// TIA Portal V17 export
// export: Created 2023-12-22T15:28:34.8526887Z, ExportSetting WithDefaults, DisplayName Totally Integrated Automation Portal, DisplayVersion V17, DisplayName TIA Portal Openness, DisplayVersion V17, DisplayName TIA Portal Version Control Interface, DisplayVersion V17, DisplayName STEP 7 Professional, DisplayVersion V17, DisplayName STEP 7 Safety, DisplayVersion V17, DisplayName WinCC Advanced, DisplayVersion V17
FUNCTION_BLOCK "DRV_V_D2A"   // FB121, LAD
TITLE = Управление клапаном с двумя дискретными положениями
{ S7_Optimized_Access := 'FALSE' }
VERSION : 0.1
// stored: AutoNumber false, IsIECCheckEnabled false, SetENOAutomatically false, UDAEnableTagReadback false
   VAR_INPUT
      All_Block : Bool;   // Аварийный останов
   END_VAR
   VAR_IN_OUT
      FB_QF : Bool;   // Защитный автомат
      FB_KM_Open : Bool;   // Пускатель - открыть
      FB_KM_Close : Bool;   // Пускатель - закрыть
      FB_Open : Bool;   // ОС - открыто
      FB_Close : Bool;   // ОС - закрыто
      S_Alarm : Bool;   // Наличие аварии
      CMD_Open : Bool;   // Команда - открыть
      CMD_Close : Bool;   // Команда - закрыть
   END_VAR
   VAR DB_SPECIFIC
      CMD : "CMD";   // Блок команд
      Mode : Int;   // Режим работы
      Status : Int;   // Статус устройства
      Use : Struct   // Функционал
         QF { S7_SetPoint := 'True'} : Bool;   // Защитный автомат
         KM_Open { S7_SetPoint := 'True'} : Bool;   // Пускатель - открыть
         KM_Close { S7_SetPoint := 'True'} : Bool;   // Пускатель - закрыть
         Open { S7_SetPoint := 'True'} : Bool := true;   // ОС - открыто
         Close { S7_SetPoint := 'True'} : Bool := true;   // ОС - закрыто
         One_KM { S7_SetPoint := 'True'} : Bool;   // Общий пускатель
         Electro { S7_SetPoint := 'True'} : Bool;   // Электропривод (остановка при срабатывании концевика)
         Cross { S7_SetPoint := 'True'} : Bool;   // Кросс-замена датчиков
         CMD_Open { S7_SetPoint := 'True'} : Bool := true;
         CMD_Close { S7_SetPoint := 'True'} : Bool;
         CMD_Reset { S7_SetPoint := 'True'} : Bool;
         calibration : Bool;
      END_STRUCT;
      FB : Struct   // Функционал
         Ready : Bool;   // Готовность к запуску
         QF : Bool;   // Защитный автомат
         KM_Open : Bool;   // Пускатель - открыть
         KM_Close : Bool;   // Пускатель - закрыть
         Open : Bool;   // ОС - открыто
         Close : Bool;   // ОС - закрыто
         Reserv : Bool;
         Local_Open : Bool;   // Локальное открытие
         Local_Close : Bool;   // Локальное закрытие
         pos_ok : Bool;   // положение достигнуто
         pos_open : Bool;   // клапан открывается
         pos_close : Bool;   // клапан закрывается
      END_STRUCT;
      ON : Bool;   // Успешно запущено
      OFF : Bool;   // Успешно остановлено
      REQ_Open : Bool;   // Запрос на открытие
      REQ_Close : Bool;   // Запрос на закрытие
   END_VAR
   VAR
      Tx { S7_SetPoint := 'True'} : Array[0..4] of "Time_S";   // Блок таймеров
   END_VAR
   VAR DB_SPECIFIC
      Inv : Struct   // Инверсия сигналов
         CMD { S7_SetPoint := 'True'} : Bool;   // Команда запуска
         QF { S7_SetPoint := 'True'} : Bool;   // Защитный автомат
         KM_Open { S7_SetPoint := 'True'} : Bool;   // Пускатель - открыть
         KM_Close { S7_SetPoint := 'True'} : Bool;   // Пускатель - закрыть
         Serivce { S7_SetPoint := 'True'} : Bool;   // Сервисный выключатель
         Open { S7_SetPoint := 'True'} : Bool;   // ОС - открыто
         Close { S7_SetPoint := 'True'} : Bool;   // ОС - закрыто
         Local_Open { S7_SetPoint := 'True'} : Bool;   // Локальное открытие
         Local_Close { S7_SetPoint := 'True'} : Bool;   // Локальное закрытие
      END_STRUCT;
      Alarm : Struct   // Список аварий
         Block : Bool;   // Аварийная остановка
         QF : Bool;   // Выбило защитный автомат
         KM_Open : Bool;   // Не сработал пускатель - открыть
         KM_Close : Bool;   // Не сработал пускатель - закрыть
         Two_S : Bool;   // Две ОС
         Open : Bool;   // Не сработал концевик - открыто
         Close : Bool;   // Не сработал концевик - закрыто
         OpTime : Bool;
      END_STRUCT;
      Alarms : Word;   // Слово аварий
      OpTime_h : DInt;   // наработка (ч)
      OpTime_s { S7_SetPoint := 'True'} : DInt;   // наработка (с)
      CodeID { S7_SetPoint := 'True'} : Int;   // Код датчика для привязки в скаде
      Indirect : Struct
         FB_QF { S7_SetPoint := 'True'} : Bool := true;   // Защитный автомат
         FB_KM_Open { S7_SetPoint := 'True'} : Bool := true;   // Пускатель - открыть
         FB_KM_Close { S7_SetPoint := 'True'} : Bool := true;   // Пускатель - закрыть
         FB_Open { S7_SetPoint := 'True'} : Bool := true;   // ОС - открыто
         FB_Close { S7_SetPoint := 'True'} : Bool := true;   // ОС - закрыто
         CMD_Open { S7_SetPoint := 'True'} : Bool := true;   // Команда на открытие
         CMD_Close { S7_SetPoint := 'True'} : Bool := true;   // Команда на закрытие
      END_STRUCT;
      Indirect_BYTE : Struct
         FB_QF { S7_SetPoint := 'True'} : Int;   // Защитный автомат
         FB_KM_Open { S7_SetPoint := 'True'} : Int;   // Пускатель - открыть
         FB_KM_Close { S7_SetPoint := 'True'} : Int;   // Пускатель - закрыть
         FB_Open { S7_SetPoint := 'True'} : Int;   // ОС - открыто
         FB_Close { S7_SetPoint := 'True'} : Int;   // ОС - закрыто
         CMD_Open { S7_SetPoint := 'True'} : Int;   // Команда на открытие
         CMD_Close { S7_SetPoint := 'True'} : Int;   // Команда на закрытие
         CMD_Reset : Int;
      END_STRUCT;
      Indirect_BIT : Struct
         FB_QF { S7_SetPoint := 'True'} : Int;   // Защитный автомат
         FB_KM_Open { S7_SetPoint := 'True'} : Int;   // Пускатель - открыть
         FB_KM_Close { S7_SetPoint := 'True'} : Int;   // Пускатель - закрыть
         FB_Open { S7_SetPoint := 'True'} : Int;   // ОС - открыто
         FB_Close { S7_SetPoint := 'True'} : Int;   // ОС - закрыто
         CMD_Open { S7_SetPoint := 'True'} : Int;   // Команда на открытие
         CMD_Close { S7_SetPoint := 'True'} : Int;   // Команда на закрытие
         CMD_Reset : Int;
      END_STRUCT;
   END_VAR
   VAR
      Tx_Sm { S7_SetPoint := 'True'} : Array[0..2] of "Time_S_b";   // Блок таймеров
      Tx_R { S7_SetPoint := 'True'} : Array[0..1] of "Time_R";   // Блок таймеров
   END_VAR
   VAR DB_SPECIFIC
      SP_A : Real;
      SP_M : Real;
      SP : Real;
      POSITION : Real;
      "step" : Int;
      DB { S7_SetPoint := 'True'} : Real := 1.0;
      pos : Array[0..15] of Bool;
   END_VAR
   VAR_TEMP
      xQF : Bool;
      xKM_Open : Bool;
      xKM_Close : Bool;
      xOpen : Bool;
      xClose : Bool;
      min : Real;
      max : Real;
   END_VAR
   VAR CONSTANT
      Pos_MIN : Real := 0.0;
      Pos_MAX : Real := 100.0;
   END_VAR
   VAR_TEMP   // added for the SCL form of the ladder/FBD networks
      _w1 : Bool;
      _w2 : Bool;
      _w3 : Bool;
      _w4 : Bool;
      _w5 : Bool;
      _w6 : Bool;
      _w7 : Bool;
   END_VAR
BEGIN

REGION Network 1: Режим глобальной симуляции
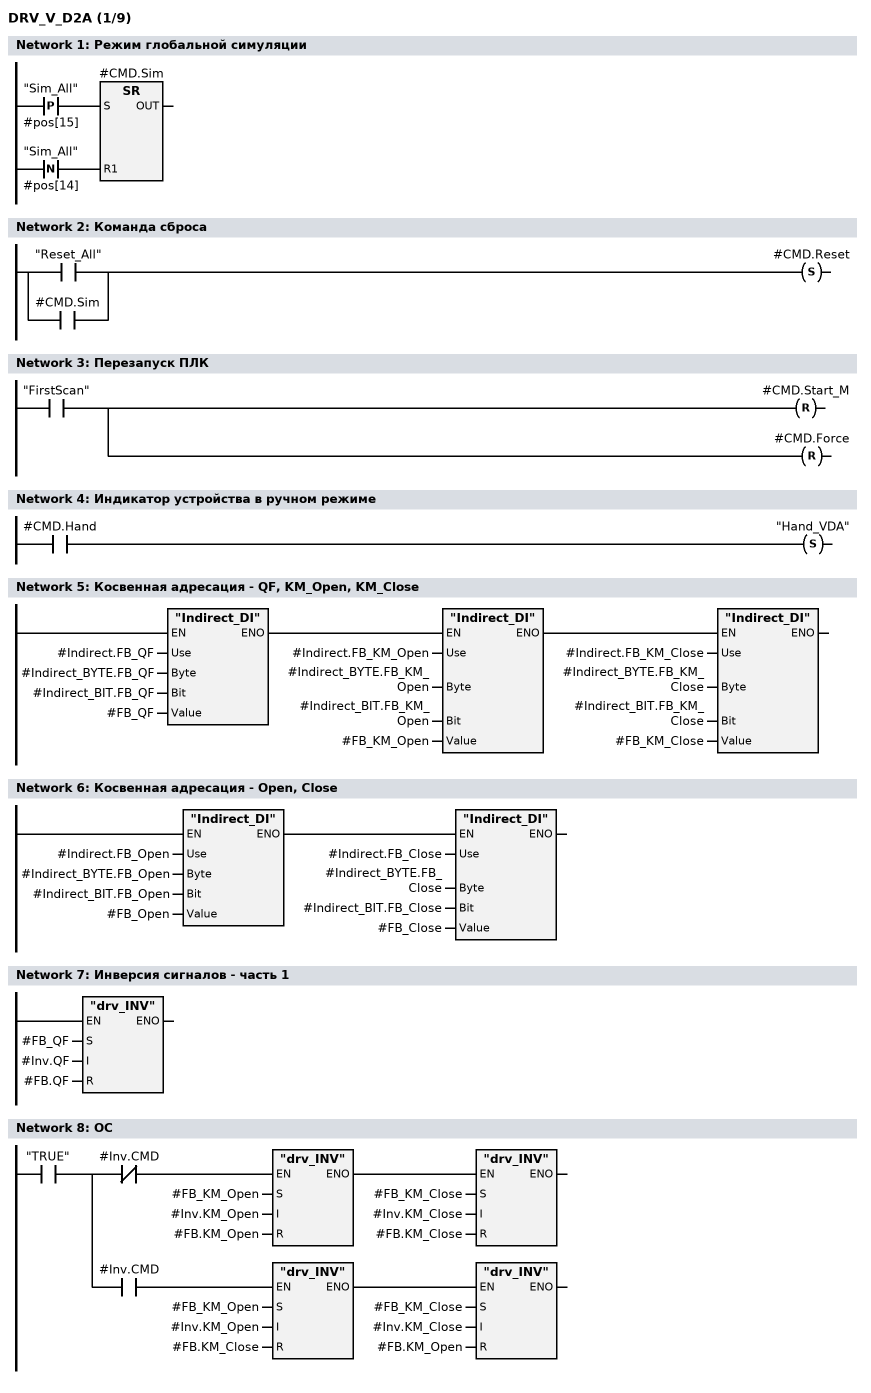
   RUNG wire#powerrail
      P_Contact(operand := "Sim_All", bit := #pos[15])
      S_SR(operand := #CMD.Sim, r1 := wire#w1)
   END_RUNG
   RUNG wire#powerrail
      N_Contact(operand := "Sim_All", bit := #pos[14])
   END_RUNG wire#w1
   // the same network as SCL:
   #_w1 := "Sim_All" AND NOT #pos[15];   // rising edge of "Sim_All"
   #pos[15] := "Sim_All";
   #_w2 := NOT "Sim_All" AND #pos[14];   // falling edge of "Sim_All"
   #pos[14] := "Sim_All";
   IF #_w1 THEN
       #CMD.Sim := TRUE;   // SR flip-flop
   END_IF;
   IF #_w2 THEN #CMD.Sim := FALSE; END_IF;
END_REGION

REGION Network 2: Команда сброса
   RUNG wire#powerrail
      Contact( "Reset_All" )
      wire#w1
      S_Coil( #CMD.Reset )
   END_RUNG
   RUNG wire#powerrail
      Contact( #CMD.Sim )
   END_RUNG wire#w1
   // the same network as SCL:
   IF "Reset_All" OR #CMD.Sim THEN #CMD.Reset := TRUE; END_IF;
END_REGION

REGION Network 3: Перезапуск ПЛК
   RUNG wire#powerrail
      Contact( "FirstScan" )
      wire#w1
      R_Coil( #CMD.Start_M )
   END_RUNG
   RUNG wire#w1
      R_Coil( #CMD.Force )
   END_RUNG
   // the same network as SCL:
   IF "FirstScan" THEN
       #CMD.Start_M := FALSE;
       #CMD.Force := FALSE;
   END_IF;
END_REGION

REGION Network 4: Индикатор устройства в ручном режиме
   RUNG wire#powerrail
      Contact( #CMD.Hand )
      S_Coil( "Hand_VDA" )
   END_RUNG
   // the same network as SCL:
   IF #CMD.Hand THEN "Hand_VDA" := TRUE; END_IF;
END_REGION

REGION Network 5: Косвенная адресация - QF, KM_Open, KM_Close
   RUNG wire#powerrail
      "Indirect_DI"(Use := #Indirect.FB_QF, "Byte" := #Indirect_BYTE.FB_QF, Bit := #Indirect_BIT.FB_QF, Value := #FB_QF)
      "Indirect_DI"(Use := #Indirect.FB_KM_Open, "Byte" := #Indirect_BYTE.FB_KM_Open, Bit := #Indirect_BIT.FB_KM_Open, Value := #FB_KM_Open)
      "Indirect_DI"(Use := #Indirect.FB_KM_Close, "Byte" := #Indirect_BYTE.FB_KM_Close, Bit := #Indirect_BIT.FB_KM_Close, Value := #FB_KM_Close)
   END_RUNG
   // the same network as SCL:
   "Indirect_DI"(Use := #Indirect.FB_QF,
                 "Byte" := #Indirect_BYTE.FB_QF,
                 Bit := #Indirect_BIT.FB_QF,
                 Value := #FB_QF,
                 ENO => #_w1);
   "Indirect_DI"(EN := #_w1,
                 Use := #Indirect.FB_KM_Open,
                 "Byte" := #Indirect_BYTE.FB_KM_Open,
                 Bit := #Indirect_BIT.FB_KM_Open,
                 Value := #FB_KM_Open,
                 ENO => #_w2);
   IF #_w2 THEN
       "Indirect_DI"(Use := #Indirect.FB_KM_Close,
                     "Byte" := #Indirect_BYTE.FB_KM_Close,
                     Bit := #Indirect_BIT.FB_KM_Close,
                     Value := #FB_KM_Close);
   END_IF;
END_REGION

REGION Network 6: Косвенная адресация - Open, Close
   RUNG wire#powerrail
      "Indirect_DI"(Use := #Indirect.FB_Open, "Byte" := #Indirect_BYTE.FB_Open, Bit := #Indirect_BIT.FB_Open, Value := #FB_Open)
      "Indirect_DI"(Use := #Indirect.FB_Close, "Byte" := #Indirect_BYTE.FB_Close, Bit := #Indirect_BIT.FB_Close, Value := #FB_Close)
   END_RUNG
   // the same network as SCL:
   "Indirect_DI"(Use := #Indirect.FB_Open,
                 "Byte" := #Indirect_BYTE.FB_Open,
                 Bit := #Indirect_BIT.FB_Open,
                 Value := #FB_Open,
                 ENO => #_w1);
   IF #_w1 THEN
       "Indirect_DI"(Use := #Indirect.FB_Close,
                     "Byte" := #Indirect_BYTE.FB_Close,
                     Bit := #Indirect_BIT.FB_Close,
                     Value := #FB_Close);
   END_IF;
END_REGION

REGION Network 7: Инверсия сигналов - часть 1
   RUNG wire#powerrail
      "drv_INV"(S := #FB_QF, I := #Inv.QF, R := #FB.QF)
   END_RUNG
   // the same network as SCL:
   "drv_INV"(S := #FB_QF, I := #Inv.QF, R := #FB.QF);
END_REGION

REGION Network 8: ОС
   RUNG wire#powerrail
      Contact( "TRUE" )
      wire#w1
      I_Contact( #Inv.CMD )
      "drv_INV"(S := #FB_KM_Open, I := #Inv.KM_Open, R := #FB.KM_Open)
      "drv_INV"(S := #FB_KM_Close, I := #Inv.KM_Close, R := #FB.KM_Close)
   END_RUNG
   RUNG wire#w1
      Contact( #Inv.CMD )
      "drv_INV"(S := #FB_KM_Open, I := #Inv.KM_Open, R := #FB.KM_Close)
      "drv_INV"(S := #FB_KM_Close, I := #Inv.KM_Close, R := #FB.KM_Open)
   END_RUNG
   // the same network as SCL:
   #_w2 := "TRUE";
   "drv_INV"(EN := "TRUE" AND NOT #Inv.CMD, S := #FB_KM_Open, I := #Inv.KM_Open, R := #FB.KM_Open, ENO => #_w1);
   IF #_w1 THEN "drv_INV"(S := #FB_KM_Close, I := #Inv.KM_Close, R := #FB.KM_Close); END_IF;
   "drv_INV"(EN := #_w2 AND #Inv.CMD, S := #FB_KM_Open, I := #Inv.KM_Open, R := #FB.KM_Close, ENO => #_w3);
   IF #_w3 THEN "drv_INV"(S := #FB_KM_Close, I := #Inv.KM_Close, R := #FB.KM_Open); END_IF;
END_REGION

REGION Network 9: Инверсия сигналов - часть 2
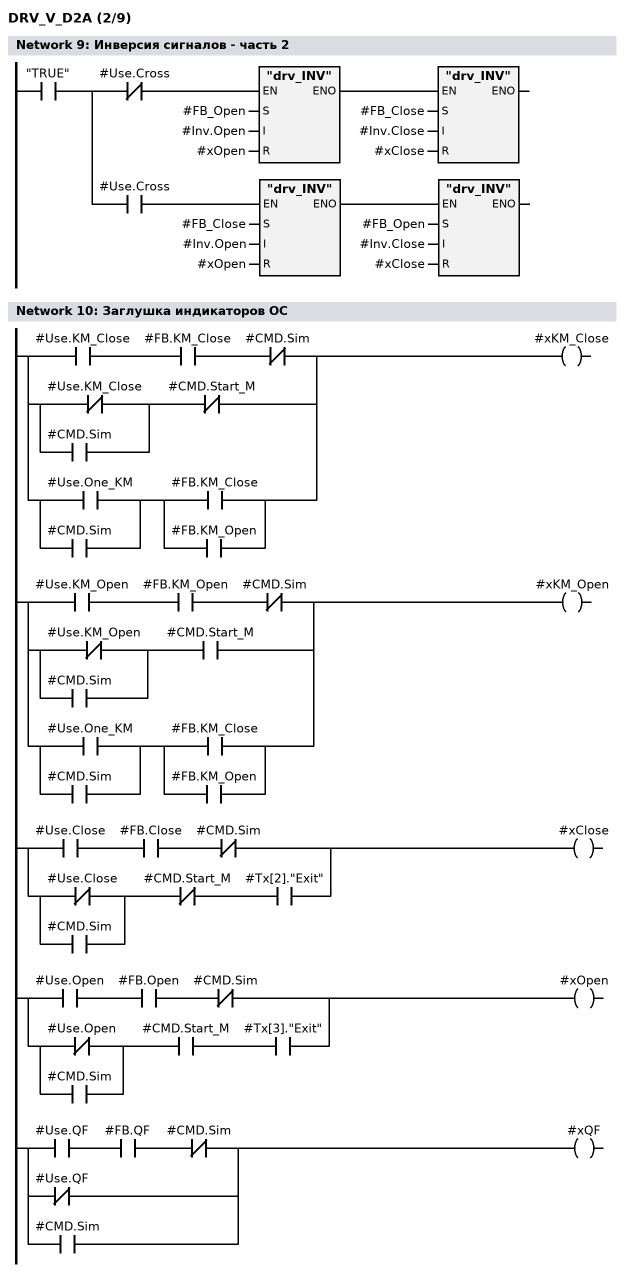
   RUNG wire#powerrail
      Contact( "TRUE" )
      wire#w1
      I_Contact( #Use.Cross )
      "drv_INV"(S := #FB_Open, I := #Inv.Open, R := #xOpen)
      "drv_INV"(S := #FB_Close, I := #Inv.Close, R := #xClose)
   END_RUNG
   RUNG wire#w1
      Contact( #Use.Cross )
      "drv_INV"(S := #FB_Close, I := #Inv.Open, R := #xOpen)
      "drv_INV"(S := #FB_Open, I := #Inv.Close, R := #xClose)
   END_RUNG
   // the same network as SCL:
   #_w2 := "TRUE";
   "drv_INV"(EN := "TRUE" AND NOT #Use.Cross, S := #FB_Open, I := #Inv.Open, R := #xOpen, ENO => #_w1);
   IF #_w1 THEN "drv_INV"(S := #FB_Close, I := #Inv.Close, R := #xClose); END_IF;
   "drv_INV"(EN := #_w2 AND #Use.Cross, S := #FB_Close, I := #Inv.Open, R := #xOpen, ENO => #_w3);
   IF #_w3 THEN "drv_INV"(S := #FB_Open, I := #Inv.Close, R := #xClose); END_IF;
END_REGION

REGION Network 10: Заглушка индикаторов ОС
   RUNG wire#powerrail
      Contact( #Use.KM_Close )
      Contact( #FB.KM_Close )
      I_Contact( #CMD.Sim )
      wire#w1
      Coil( #xKM_Close )
   END_RUNG
   RUNG wire#powerrail
      I_Contact( #Use.KM_Close )
      wire#w2
      I_Contact( #CMD.Start_M )
   END_RUNG wire#w1
   RUNG wire#powerrail
      Contact( #CMD.Sim )
   END_RUNG wire#w2
   RUNG wire#powerrail
      Contact( #Use.One_KM )
      wire#w3
      Contact( #FB.KM_Close )
   END_RUNG wire#w1
   RUNG wire#powerrail
      Contact( #CMD.Sim )
   END_RUNG wire#w3
   RUNG wire#w3
      Contact( #FB.KM_Open )
   END_RUNG wire#w1
   RUNG wire#powerrail
      Contact( #Use.KM_Open )
      Contact( #FB.KM_Open )
      I_Contact( #CMD.Sim )
      wire#w4
      Coil( #xKM_Open )
   END_RUNG
   RUNG wire#powerrail
      I_Contact( #Use.KM_Open )
      wire#w5
      Contact( #CMD.Start_M )
   END_RUNG wire#w4
   RUNG wire#powerrail
      Contact( #CMD.Sim )
   END_RUNG wire#w5
   RUNG wire#powerrail
      Contact( #Use.One_KM )
      wire#w6
      Contact( #FB.KM_Close )
   END_RUNG wire#w4
   RUNG wire#powerrail
      Contact( #CMD.Sim )
   END_RUNG wire#w6
   RUNG wire#w6
      Contact( #FB.KM_Open )
   END_RUNG wire#w4
   RUNG wire#powerrail
      Contact( #Use.Close )
      Contact( #FB.Close )
      I_Contact( #CMD.Sim )
      wire#w7
      Coil( #xClose )
   END_RUNG
   RUNG wire#powerrail
      I_Contact( #Use.Close )
      wire#w8
      I_Contact( #CMD.Start_M )
      Contact( #Tx[2]."Exit" )
   END_RUNG wire#w7
   RUNG wire#powerrail
      Contact( #CMD.Sim )
   END_RUNG wire#w8
   RUNG wire#powerrail
      Contact( #Use.Open )
      Contact( #FB.Open )
      I_Contact( #CMD.Sim )
      wire#w9
      Coil( #xOpen )
   END_RUNG
   RUNG wire#powerrail
      I_Contact( #Use.Open )
      wire#w10
      Contact( #CMD.Start_M )
      Contact( #Tx[3]."Exit" )
   END_RUNG wire#w9
   RUNG wire#powerrail
      Contact( #CMD.Sim )
   END_RUNG wire#w10
   RUNG wire#powerrail
      Contact( #Use.QF )
      Contact( #FB.QF )
      I_Contact( #CMD.Sim )
      wire#w11
      Coil( #xQF )
   END_RUNG
   RUNG wire#powerrail
      I_Contact( #Use.QF )
   END_RUNG wire#w11
   RUNG wire#powerrail
      Contact( #CMD.Sim )
   END_RUNG wire#w11
   // the same network as SCL:
   #xKM_Close := (#Use.KM_Close AND #FB.KM_Close AND NOT #CMD.Sim) OR ((NOT #Use.KM_Close OR #CMD.Sim) AND NOT #CMD.Start_M) OR ((#Use.One_KM OR #CMD.Sim) AND (#FB.KM_Close OR #FB.KM_Open));
   #xKM_Open := (#Use.KM_Open AND #FB.KM_Open AND NOT #CMD.Sim) OR ((NOT #Use.KM_Open OR #CMD.Sim) AND #CMD.Start_M) OR ((#Use.One_KM OR #CMD.Sim) AND (#FB.KM_Close OR #FB.KM_Open));
   #xClose := (#Use.Close AND #FB.Close AND NOT #CMD.Sim) OR ((NOT #Use.Close OR #CMD.Sim) AND NOT #CMD.Start_M AND #Tx[2]."Exit");
   #xOpen := (#Use.Open AND #FB.Open AND NOT #CMD.Sim) OR ((NOT #Use.Open OR #CMD.Sim) AND #CMD.Start_M AND #Tx[3]."Exit");
   #xQF := (#Use.QF AND #FB.QF AND NOT #CMD.Sim) OR NOT #Use.QF OR #CMD.Sim;
END_REGION

REGION Network 11: Запуск
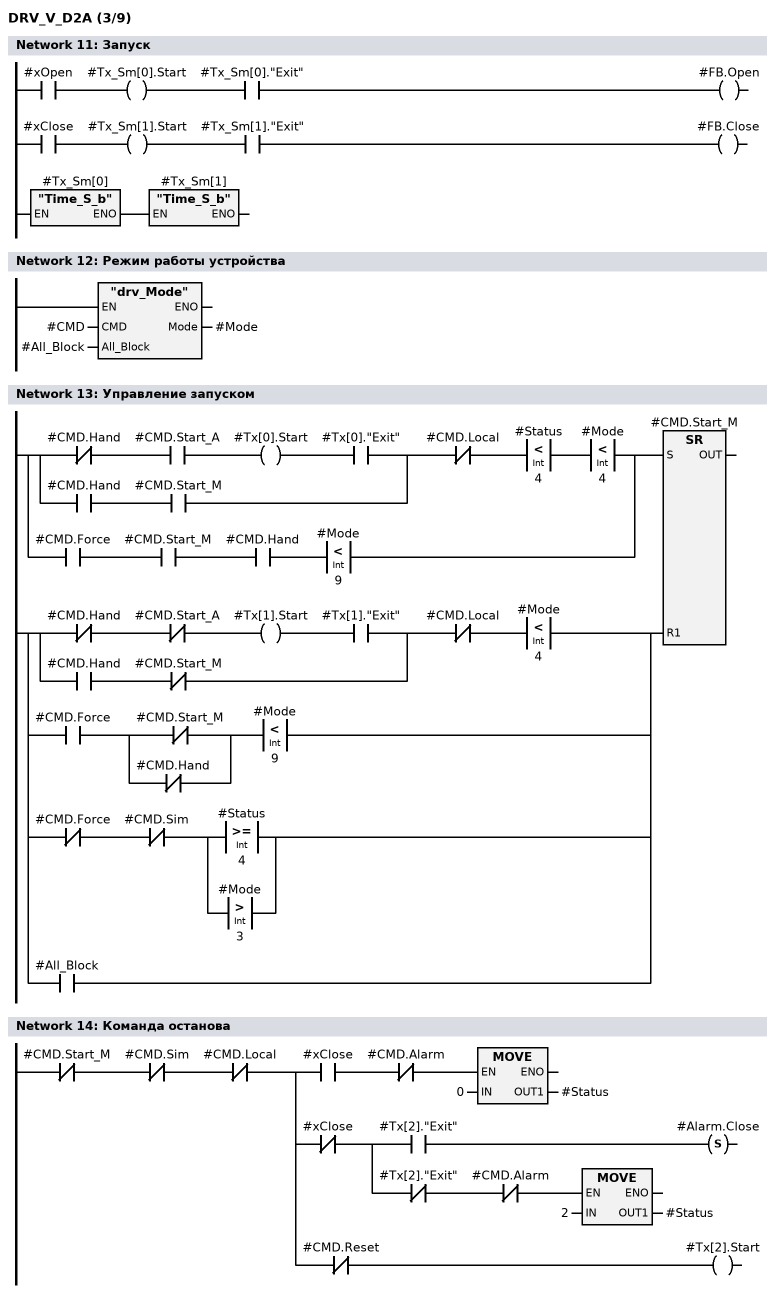
   RUNG wire#powerrail
      Contact( #xOpen )
      Coil( #Tx_Sm[0].Start )
      Contact( #Tx_Sm[0]."Exit" )
      Coil( #FB.Open )
   END_RUNG
   RUNG wire#powerrail
      Contact( #xClose )
      Coil( #Tx_Sm[1].Start )
      Contact( #Tx_Sm[1]."Exit" )
      Coil( #FB.Close )
   END_RUNG
   RUNG wire#powerrail
      #Tx_Sm[0]()
      #Tx_Sm[1]()
   END_RUNG
   // the same network as SCL:
   #Tx_Sm[0].Start := #xOpen;
   #FB.Open := #xOpen AND #Tx_Sm[0]."Exit";
   #Tx_Sm[1].Start := #xClose;
   #FB.Close := #xClose AND #Tx_Sm[1]."Exit";
   #Tx_Sm[0](ENO => #_w1);   // "Time_S_b"
   IF #_w1 THEN
       #Tx_Sm[1]();   // "Time_S_b"
   END_IF;
END_REGION

REGION Network 12: Режим работы устройства
   RUNG wire#powerrail
      "drv_Mode"(CMD := #CMD, All_Block := #All_Block, Mode => #Mode)
   END_RUNG
   // the same network as SCL:
   "drv_Mode"(CMD := #CMD, All_Block := #All_Block, Mode => #Mode);
END_REGION

REGION Network 13: Управление запуском
   RUNG wire#powerrail
      I_Contact( #CMD.Hand )
      Contact( #CMD.Start_A )
      Coil( #Tx[0].Start )
      Contact( #Tx[0]."Exit" )
      wire#w1
      I_Contact( #CMD.Local )
      { S7_Templates := "SrcType := Int" } LT_Contact(in1 := #Status, in2 := 4)
      { S7_Templates := "SrcType := Int" } LT_Contact(in1 := #Mode, in2 := 4)
      wire#w2
      S_SR(operand := #CMD.Start_M, r1 := wire#w7)
   END_RUNG
   RUNG wire#powerrail
      Contact( #CMD.Hand )
      Contact( #CMD.Start_M )
   END_RUNG wire#w1
   RUNG wire#powerrail
      Contact( #CMD.Force )
      Contact( #CMD.Start_M )
      Contact( #CMD.Hand )
      { S7_Templates := "SrcType := Int" } LT_Contact(in1 := #Mode, in2 := 9)
   END_RUNG wire#w2
   RUNG wire#powerrail
      I_Contact( #CMD.Hand )
      I_Contact( #CMD.Start_A )
      Coil( #Tx[1].Start )
      Contact( #Tx[1]."Exit" )
      wire#w3
      I_Contact( #CMD.Local )
      { S7_Templates := "SrcType := Int" } LT_Contact(in1 := #Mode, in2 := 4)
   END_RUNG wire#w7
   RUNG wire#powerrail
      Contact( #CMD.Hand )
      I_Contact( #CMD.Start_M )
   END_RUNG wire#w3
   RUNG wire#powerrail
      Contact( #CMD.Force )
      wire#w4
      I_Contact( #CMD.Start_M )
      wire#w5
      { S7_Templates := "SrcType := Int" } LT_Contact(in1 := #Mode, in2 := 9)
   END_RUNG wire#w7
   RUNG wire#w4
      I_Contact( #CMD.Hand )
   END_RUNG wire#w5
   RUNG wire#powerrail
      I_Contact( #CMD.Force )
      I_Contact( #CMD.Sim )
      wire#w6
      { S7_Templates := "SrcType := Int" } GE_Contact(in1 := #Status, in2 := 4)
   END_RUNG wire#w7
   RUNG wire#w6
      { S7_Templates := "SrcType := Int" } GT_Contact(in1 := #Mode, in2 := 3)
   END_RUNG wire#w7
   RUNG wire#powerrail
      Contact( #All_Block )
   END_RUNG wire#w7
   // the same network as SCL:
   #Tx[0].Start := NOT #CMD.Hand AND #CMD.Start_A;
   #_w1 := (((NOT #CMD.Hand AND #CMD.Start_A AND #Tx[0]."Exit") OR (#CMD.Hand AND #CMD.Start_M)) AND NOT #CMD.Local AND (#Status < 4) AND (#Mode < 4)) OR (#CMD.Force AND #CMD.Start_M AND #CMD.Hand AND (#Mode < 9));
   #Tx[1].Start := NOT #CMD.Hand AND NOT #CMD.Start_A;
   #_w2 := (((NOT #CMD.Hand AND NOT #CMD.Start_A AND #Tx[1]."Exit") OR (#CMD.Hand AND NOT #CMD.Start_M)) AND NOT #CMD.Local AND (#Mode < 4)) OR (#CMD.Force AND (NOT #CMD.Start_M OR NOT #CMD.Hand) AND (#Mode < 9)) OR (NOT #CMD.Force AND NOT #CMD.Sim AND ((#Status >= 4) OR (#Mode > 3))) OR #All_Block;
   IF #_w1 THEN
       #CMD.Start_M := TRUE;   // SR flip-flop
   END_IF;
   IF #_w2 THEN #CMD.Start_M := FALSE; END_IF;
END_REGION

REGION Network 14: Команда останова
   RUNG wire#powerrail
      I_Contact( #CMD.Start_M )
      I_Contact( #CMD.Sim )
      I_Contact( #CMD.Local )
      wire#w1
      Contact( #xClose )
      I_Contact( #CMD.Alarm )
      { S7_GenerateENO := "TRUE" } Move(in := 0, out1 => #Status)
   END_RUNG
   RUNG wire#w1
      I_Contact( #xClose )
      wire#w2
      Contact( #Tx[2]."Exit" )
      S_Coil( #Alarm.Close )
   END_RUNG
   RUNG wire#w2
      I_Contact( #Tx[2]."Exit" )
      I_Contact( #CMD.Alarm )
      { S7_GenerateENO := "TRUE" } Move(in := 2, out1 => #Status)
   END_RUNG
   RUNG wire#w1
      I_Contact( #CMD.Reset )
      Coil( #Tx[2].Start )
   END_RUNG
   // the same network as SCL:
   #_w1 := NOT #CMD.Start_M AND NOT #CMD.Sim AND NOT #CMD.Local;
   IF #_w1 AND #xClose AND NOT #CMD.Alarm THEN #Status := 0; END_IF;
   #_w2 := #_w1 AND NOT #xClose;
   IF #_w2 AND #Tx[2]."Exit" THEN #Alarm.Close := TRUE; END_IF;
   IF #_w2 AND NOT #Tx[2]."Exit" AND NOT #CMD.Alarm THEN #Status := 2; END_IF;
   #Tx[2].Start := #_w1 AND NOT #CMD.Reset;
END_REGION

REGION Network 15: Команда запуска
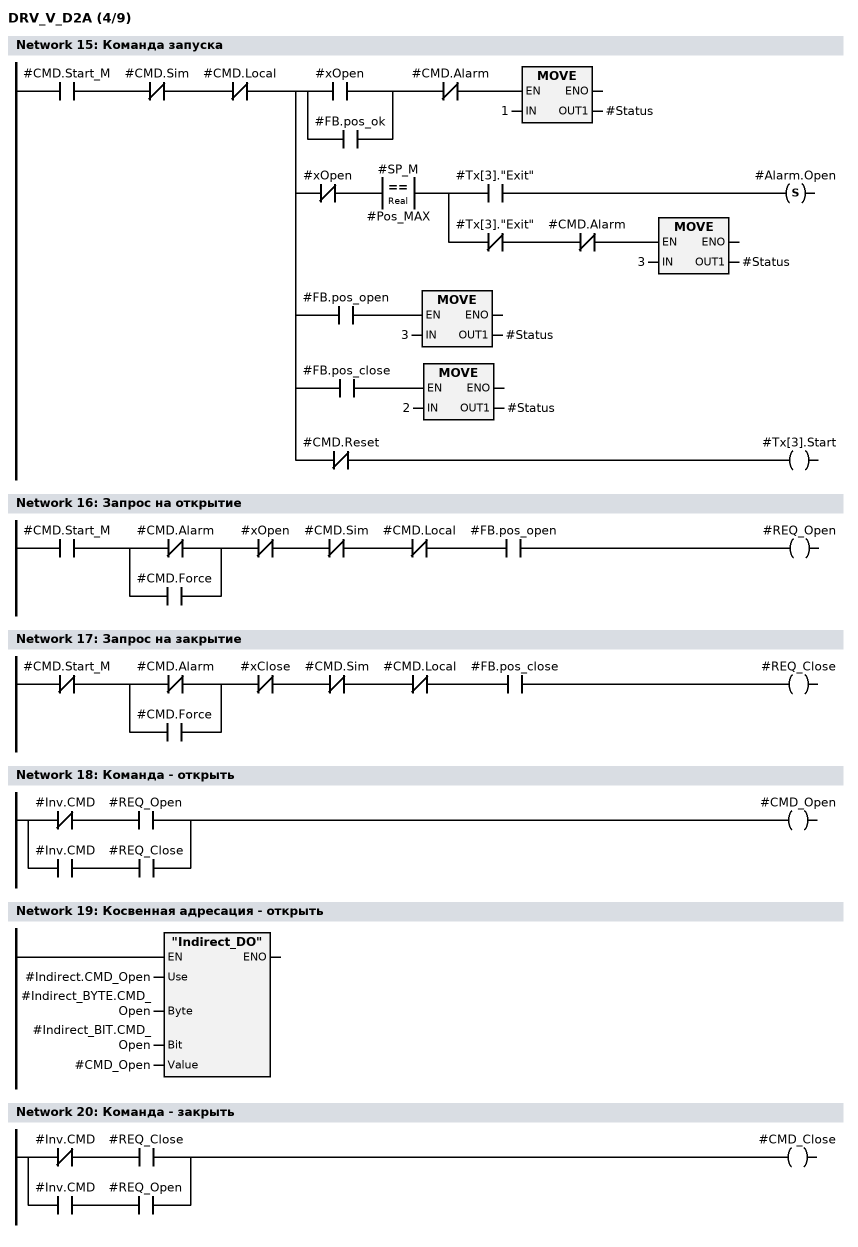
   RUNG wire#powerrail
      Contact( #CMD.Start_M )
      I_Contact( #CMD.Sim )
      I_Contact( #CMD.Local )
      wire#w1
      Contact( #xOpen )
      wire#w2
      I_Contact( #CMD.Alarm )
      { S7_GenerateENO := "TRUE" } Move(in := 1, out1 => #Status)
   END_RUNG
   RUNG wire#w1
      Contact( #FB.pos_ok )
   END_RUNG wire#w2
   RUNG wire#w1
      I_Contact( #xOpen )
      { S7_Templates := "SrcType := Real" } EQ_Contact(in1 := #SP_M, in2 := #Pos_MAX)
      wire#w3
      Contact( #Tx[3]."Exit" )
      S_Coil( #Alarm.Open )
   END_RUNG
   RUNG wire#w3
      I_Contact( #Tx[3]."Exit" )
      I_Contact( #CMD.Alarm )
      { S7_GenerateENO := "TRUE" } Move(in := 3, out1 => #Status)
   END_RUNG
   RUNG wire#w1
      Contact( #FB.pos_open )
      { S7_GenerateENO := "TRUE" } Move(in := 3, out1 => #Status)
   END_RUNG
   RUNG wire#w1
      Contact( #FB.pos_close )
      { S7_GenerateENO := "TRUE" } Move(in := 2, out1 => #Status)
   END_RUNG
   RUNG wire#w1
      I_Contact( #CMD.Reset )
      Coil( #Tx[3].Start )
   END_RUNG
   // the same network as SCL:
   #_w1 := #CMD.Start_M AND NOT #CMD.Sim AND NOT #CMD.Local;
   IF #_w1 AND (#xOpen OR #FB.pos_ok) AND NOT #CMD.Alarm THEN #Status := 1; END_IF;
   #_w2 := #_w1 AND NOT #xOpen AND (#SP_M = #Pos_MAX);
   IF #_w2 AND #Tx[3]."Exit" THEN #Alarm.Open := TRUE; END_IF;
   IF #_w2 AND NOT #Tx[3]."Exit" AND NOT #CMD.Alarm THEN #Status := 3; END_IF;
   IF #_w1 AND #FB.pos_open THEN #Status := 3; END_IF;
   IF #_w1 AND #FB.pos_close THEN #Status := 2; END_IF;
   #Tx[3].Start := #_w1 AND NOT #CMD.Reset;
END_REGION

REGION Network 16: Запрос на открытие
   RUNG wire#powerrail
      Contact( #CMD.Start_M )
      wire#w1
      I_Contact( #CMD.Alarm )
      wire#w2
      I_Contact( #xOpen )
      I_Contact( #CMD.Sim )
      I_Contact( #CMD.Local )
      Contact( #FB.pos_open )
      Coil( #REQ_Open )
   END_RUNG
   RUNG wire#w1
      Contact( #CMD.Force )
   END_RUNG wire#w2
   // the same network as SCL:
   #REQ_Open := #CMD.Start_M AND (NOT #CMD.Alarm OR #CMD.Force) AND NOT #xOpen AND NOT #CMD.Sim AND NOT #CMD.Local AND #FB.pos_open;
END_REGION

REGION Network 17: Запрос на закрытие
   RUNG wire#powerrail
      I_Contact( #CMD.Start_M )
      wire#w1
      I_Contact( #CMD.Alarm )
      wire#w2
      I_Contact( #xClose )
      I_Contact( #CMD.Sim )
      I_Contact( #CMD.Local )
      Contact( #FB.pos_close )
      Coil( #REQ_Close )
   END_RUNG
   RUNG wire#w1
      Contact( #CMD.Force )
   END_RUNG wire#w2
   // the same network as SCL:
   #REQ_Close := NOT #CMD.Start_M AND (NOT #CMD.Alarm OR #CMD.Force) AND NOT #xClose AND NOT #CMD.Sim AND NOT #CMD.Local AND #FB.pos_close;
END_REGION

REGION Network 18: Команда - открыть
   RUNG wire#powerrail
      I_Contact( #Inv.CMD )
      Contact( #REQ_Open )
      wire#w1
      Coil( #CMD_Open )
   END_RUNG
   RUNG wire#powerrail
      Contact( #Inv.CMD )
      Contact( #REQ_Close )
   END_RUNG wire#w1
   // the same network as SCL:
   #CMD_Open := (NOT #Inv.CMD AND #REQ_Open) OR (#Inv.CMD AND #REQ_Close);
END_REGION

REGION Network 19: Косвенная адресация - открыть
   RUNG wire#powerrail
      "Indirect_DO"(Use := #Indirect.CMD_Open, "Byte" := #Indirect_BYTE.CMD_Open, Bit := #Indirect_BIT.CMD_Open, Value := #CMD_Open)
   END_RUNG
   // the same network as SCL:
   "Indirect_DO"(Use := #Indirect.CMD_Open,
                 "Byte" := #Indirect_BYTE.CMD_Open,
                 Bit := #Indirect_BIT.CMD_Open,
                 Value := #CMD_Open);
END_REGION

REGION Network 20: Команда - закрыть
   RUNG wire#powerrail
      I_Contact( #Inv.CMD )
      Contact( #REQ_Close )
      wire#w1
      Coil( #CMD_Close )
   END_RUNG
   RUNG wire#powerrail
      Contact( #Inv.CMD )
      Contact( #REQ_Open )
   END_RUNG wire#w1
   // the same network as SCL:
   #CMD_Close := (NOT #Inv.CMD AND #REQ_Close) OR (#Inv.CMD AND #REQ_Open);
END_REGION

REGION Network 21: Косвенная адресация - закрыть
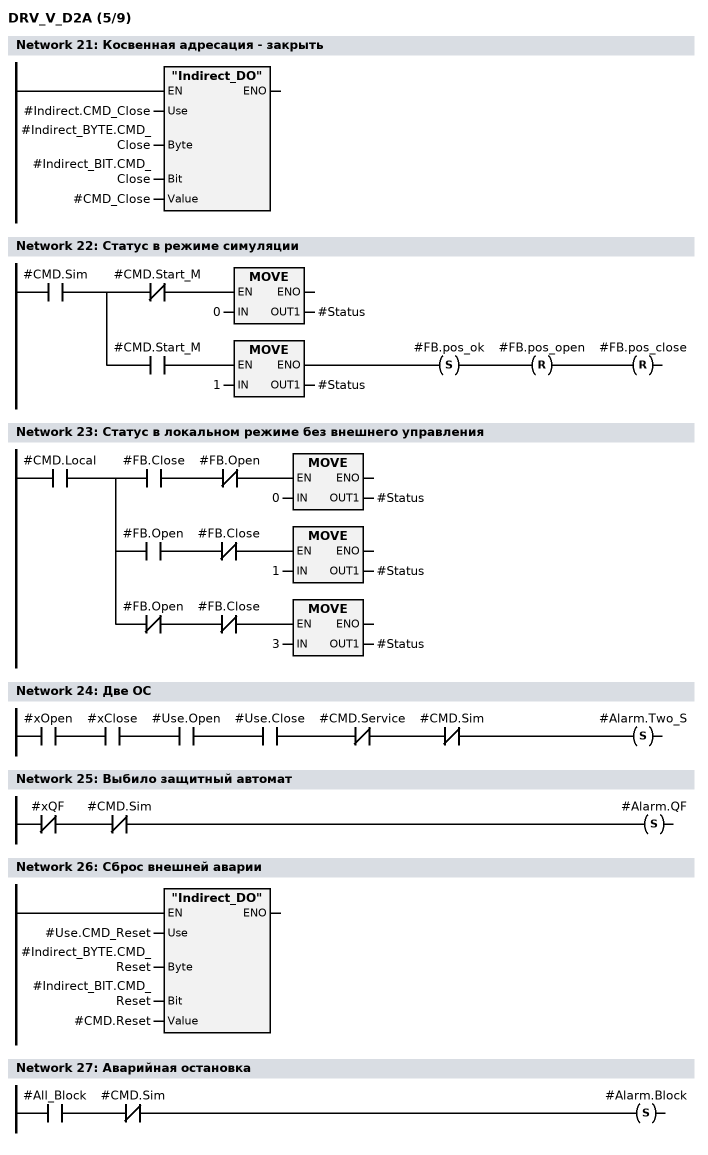
   RUNG wire#powerrail
      "Indirect_DO"(Use := #Indirect.CMD_Close, "Byte" := #Indirect_BYTE.CMD_Close, Bit := #Indirect_BIT.CMD_Close, Value := #CMD_Close)
   END_RUNG
   // the same network as SCL:
   "Indirect_DO"(Use := #Indirect.CMD_Close,
                 "Byte" := #Indirect_BYTE.CMD_Close,
                 Bit := #Indirect_BIT.CMD_Close,
                 Value := #CMD_Close);
END_REGION

REGION Network 22: Статус в режиме симуляции
   RUNG wire#powerrail
      Contact( #CMD.Sim )
      wire#w1
      I_Contact( #CMD.Start_M )
      { S7_GenerateENO := "TRUE" } Move(in := 0, out1 => #Status)
   END_RUNG
   RUNG wire#w1
      Contact( #CMD.Start_M )
      { S7_GenerateENO := "TRUE" } Move(in := 1, out1 => #Status)
      S_Coil( #FB.pos_ok )
      R_Coil( #FB.pos_open )
      R_Coil( #FB.pos_close )
   END_RUNG
   // the same network as SCL:
   // ENO of a box is taken as its EN; it also drops when the box reports an error
   IF #CMD.Sim AND NOT #CMD.Start_M THEN #Status := 0; END_IF;
   IF #CMD.Sim AND #CMD.Start_M THEN
       #Status := 1;
       #FB.pos_ok := TRUE;
       #FB.pos_open := FALSE;
       #FB.pos_close := FALSE;
   END_IF;
END_REGION

REGION Network 23: Статус в локальном режиме без внешнего управления
   RUNG wire#powerrail
      Contact( #CMD.Local )
      wire#w1
      Contact( #FB.Close )
      I_Contact( #FB.Open )
      { S7_GenerateENO := "TRUE" } Move(in := 0, out1 => #Status)
   END_RUNG
   RUNG wire#w1
      Contact( #FB.Open )
      I_Contact( #FB.Close )
      { S7_GenerateENO := "TRUE" } Move(in := 1, out1 => #Status)
   END_RUNG
   RUNG wire#w1
      I_Contact( #FB.Open )
      I_Contact( #FB.Close )
      { S7_GenerateENO := "TRUE" } Move(in := 3, out1 => #Status)
   END_RUNG
   // the same network as SCL:
   IF #CMD.Local AND #FB.Close AND NOT #FB.Open THEN #Status := 0; END_IF;
   IF #CMD.Local AND #FB.Open AND NOT #FB.Close THEN #Status := 1; END_IF;
   IF #CMD.Local AND NOT #FB.Open AND NOT #FB.Close THEN #Status := 3; END_IF;
END_REGION

REGION Network 24: Две ОС
   RUNG wire#powerrail
      Contact( #xOpen )
      Contact( #xClose )
      Contact( #Use.Open )
      Contact( #Use.Close )
      I_Contact( #CMD.Service )
      I_Contact( #CMD.Sim )
      S_Coil( #Alarm.Two_S )
   END_RUNG
   // the same network as SCL:
   IF #xOpen AND #xClose AND #Use.Open AND #Use.Close AND NOT #CMD.Service AND NOT #CMD.Sim THEN
       #Alarm.Two_S := TRUE;
   END_IF;
END_REGION

REGION Network 25: Выбило защитный автомат
   RUNG wire#powerrail
      I_Contact( #xQF )
      I_Contact( #CMD.Sim )
      S_Coil( #Alarm.QF )
   END_RUNG
   // the same network as SCL:
   IF NOT #xQF AND NOT #CMD.Sim THEN #Alarm.QF := TRUE; END_IF;
END_REGION

REGION Network 26: Сброс внешней аварии
   RUNG wire#powerrail
      "Indirect_DO"(Use := #Use.CMD_Reset, "Byte" := #Indirect_BYTE.CMD_Reset, Bit := #Indirect_BIT.CMD_Reset, Value := #CMD.Reset)
   END_RUNG
   // the same network as SCL:
   "Indirect_DO"(Use := #Use.CMD_Reset,
                 "Byte" := #Indirect_BYTE.CMD_Reset,
                 Bit := #Indirect_BIT.CMD_Reset,
                 Value := #CMD.Reset);
END_REGION

REGION Network 27: Аварийная остановка
   RUNG wire#powerrail
      Contact( #All_Block )
      I_Contact( #CMD.Sim )
      S_Coil( #Alarm.Block )
   END_RUNG
   // the same network as SCL:
   IF #All_Block AND NOT #CMD.Sim THEN #Alarm.Block := TRUE; END_IF;
END_REGION

REGION Network 28: Авария
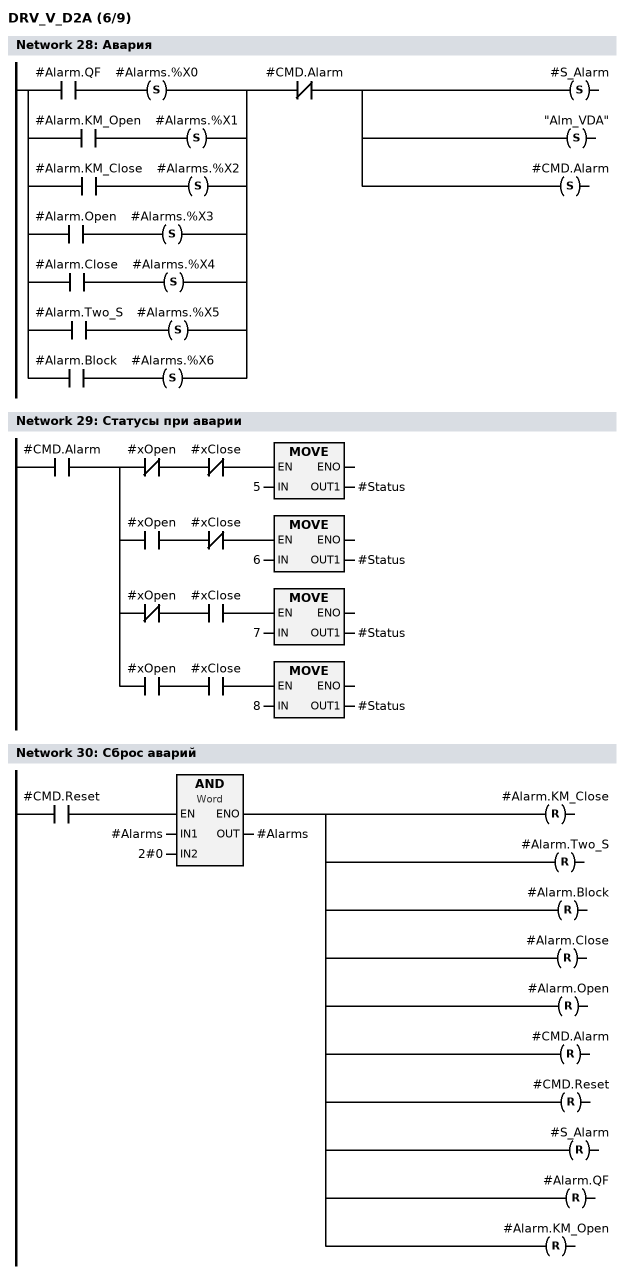
   RUNG wire#powerrail
      Contact( #Alarm.QF )
      S_Coil( #Alarms.%X0 )
      wire#w1
      I_Contact( #CMD.Alarm )
      wire#w2
      S_Coil( #S_Alarm )
   END_RUNG
   RUNG wire#powerrail
      Contact( #Alarm.KM_Open )
      S_Coil( #Alarms.%X1 )
   END_RUNG wire#w1
   RUNG wire#powerrail
      Contact( #Alarm.KM_Close )
      S_Coil( #Alarms.%X2 )
   END_RUNG wire#w1
   RUNG wire#powerrail
      Contact( #Alarm.Open )
      S_Coil( #Alarms.%X3 )
   END_RUNG wire#w1
   RUNG wire#powerrail
      Contact( #Alarm.Close )
      S_Coil( #Alarms.%X4 )
   END_RUNG wire#w1
   RUNG wire#powerrail
      Contact( #Alarm.Two_S )
      S_Coil( #Alarms.%X5 )
   END_RUNG wire#w1
   RUNG wire#powerrail
      Contact( #Alarm.Block )
      S_Coil( #Alarms.%X6 )
   END_RUNG wire#w1
   RUNG wire#w2
      S_Coil( "Alm_VDA" )
   END_RUNG
   RUNG wire#w2
      S_Coil( #CMD.Alarm )
   END_RUNG
   // the same network as SCL:
   IF #Alarm.QF THEN #Alarms.%X0 := TRUE; END_IF;
   IF #Alarm.KM_Open THEN #Alarms.%X1 := TRUE; END_IF;
   IF #Alarm.KM_Close THEN #Alarms.%X2 := TRUE; END_IF;
   IF #Alarm.Open THEN #Alarms.%X3 := TRUE; END_IF;
   IF #Alarm.Close THEN #Alarms.%X4 := TRUE; END_IF;
   IF #Alarm.Two_S THEN #Alarms.%X5 := TRUE; END_IF;
   IF #Alarm.Block THEN #Alarms.%X6 := TRUE; END_IF;
   IF (#Alarm.QF OR #Alarm.KM_Open OR #Alarm.KM_Close OR #Alarm.Open OR #Alarm.Close OR #Alarm.Two_S OR #Alarm.Block) AND NOT #CMD.Alarm THEN
       #S_Alarm := TRUE;
       "Alm_VDA" := TRUE;
       #CMD.Alarm := TRUE;
   END_IF;
END_REGION

REGION Network 29: Статусы при аварии
   RUNG wire#powerrail
      Contact( #CMD.Alarm )
      wire#w1
      I_Contact( #xOpen )
      I_Contact( #xClose )
      Move(in := 5, out1 => #Status)
   END_RUNG
   RUNG wire#w1
      Contact( #xOpen )
      I_Contact( #xClose )
      Move(in := 6, out1 => #Status)
   END_RUNG
   RUNG wire#w1
      I_Contact( #xOpen )
      Contact( #xClose )
      Move(in := 7, out1 => #Status)
   END_RUNG
   RUNG wire#w1
      Contact( #xOpen )
      Contact( #xClose )
      Move(in := 8, out1 => #Status)
   END_RUNG
   // the same network as SCL:
   IF #CMD.Alarm AND NOT #xOpen AND NOT #xClose THEN #Status := 5; END_IF;
   IF #CMD.Alarm AND #xOpen AND NOT #xClose THEN #Status := 6; END_IF;
   IF #CMD.Alarm AND NOT #xOpen AND #xClose THEN #Status := 7; END_IF;
   IF #CMD.Alarm AND #xOpen AND #xClose THEN #Status := 8; END_IF;
END_REGION

REGION Network 30: Сброс аварий
   RUNG wire#powerrail
      Contact( #CMD.Reset )
      { S7_Templates := "SrcType := Word"; S7_GenerateENO := "TRUE" } And(in1 := #Alarms, in2 := 2#0, out => #Alarms)
      wire#w1
      R_Coil( #Alarm.KM_Close )
   END_RUNG
   RUNG wire#w1
      R_Coil( #Alarm.Two_S )
   END_RUNG
   RUNG wire#w1
      R_Coil( #Alarm.Block )
   END_RUNG
   RUNG wire#w1
      R_Coil( #Alarm.Close )
   END_RUNG
   RUNG wire#w1
      R_Coil( #Alarm.Open )
   END_RUNG
   RUNG wire#w1
      R_Coil( #CMD.Alarm )
   END_RUNG
   RUNG wire#w1
      R_Coil( #CMD.Reset )
   END_RUNG
   RUNG wire#w1
      R_Coil( #S_Alarm )
   END_RUNG
   RUNG wire#w1
      R_Coil( #Alarm.QF )
   END_RUNG
   RUNG wire#w1
      R_Coil( #Alarm.KM_Open )
   END_RUNG
   // the same network as SCL:
   IF #CMD.Reset THEN
       #Alarms := #Alarms AND 2#0;
       #Alarm.KM_Close := FALSE;
       #Alarm.Two_S := FALSE;
       #Alarm.Block := FALSE;
       #Alarm.Close := FALSE;
       #Alarm.Open := FALSE;
       #CMD.Alarm := FALSE;
   END_IF;
   #_w1 := #CMD.Reset;
   IF #_w1 THEN
       #CMD.Reset := FALSE;
       #S_Alarm := FALSE;
       #Alarm.QF := FALSE;
       #Alarm.KM_Open := FALSE;
   END_IF;
END_REGION

REGION Network 31: Успешно открыто
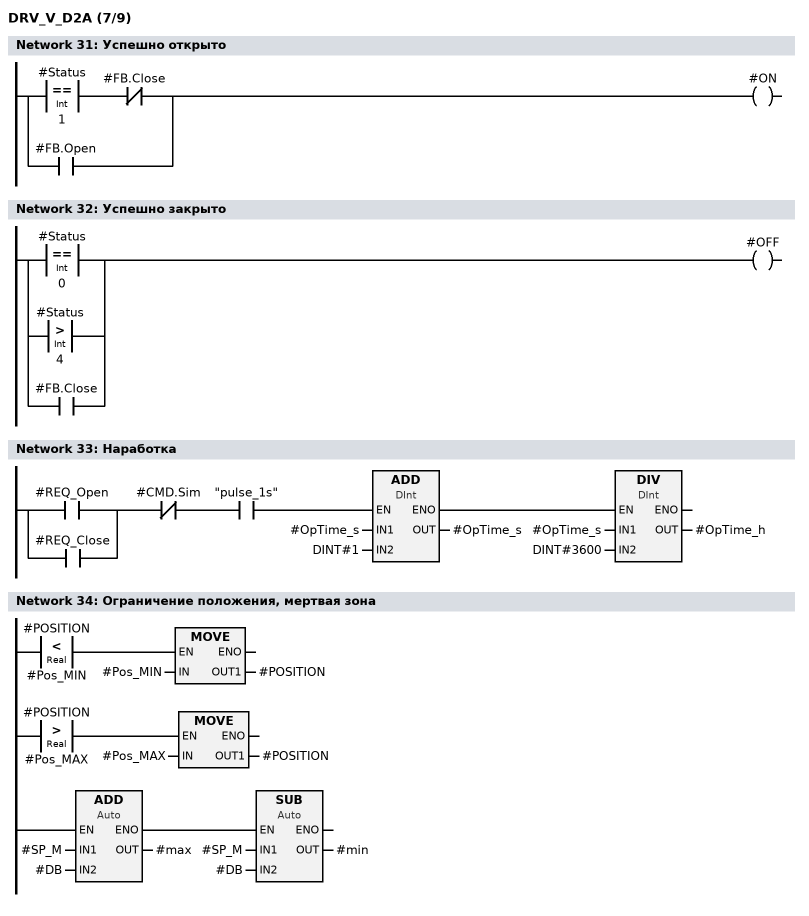
   RUNG wire#powerrail
      { S7_Templates := "SrcType := Int" } EQ_Contact(in1 := #Status, in2 := 1)
      I_Contact( #FB.Close )
      wire#w1
      Coil( #ON )
   END_RUNG
   RUNG wire#powerrail
      Contact( #FB.Open )
   END_RUNG wire#w1
   // the same network as SCL:
   #ON := ((#Status = 1) AND NOT #FB.Close) OR #FB.Open;
END_REGION

REGION Network 32: Успешно закрыто
   RUNG wire#powerrail
      { S7_Templates := "SrcType := Int" } EQ_Contact(in1 := #Status, in2 := 0)
      wire#w1
      Coil( #OFF )
   END_RUNG
   RUNG wire#powerrail
      { S7_Templates := "SrcType := Int" } GT_Contact(in1 := #Status, in2 := 4)
   END_RUNG wire#w1
   RUNG wire#powerrail
      Contact( #FB.Close )
   END_RUNG wire#w1
   // the same network as SCL:
   #OFF := (#Status = 0) OR (#Status > 4) OR #FB.Close;
END_REGION

REGION Network 33: Наработка
   RUNG wire#powerrail
      Contact( #REQ_Open )
      wire#w1
      I_Contact( #CMD.Sim )
      Contact( "pulse_1s" )
      { S7_Templates := "SrcType := DInt"; S7_GenerateENO := "TRUE" } Add(in1 := #OpTime_s, in2 := DINT#1, out => #OpTime_s)
      { S7_Templates := "SrcType := DInt"; S7_GenerateENO := "TRUE" } Div(in1 := #OpTime_s, in2 := DINT#3600, out => #OpTime_h)
   END_RUNG
   RUNG wire#powerrail
      Contact( #REQ_Close )
   END_RUNG wire#w1
   // the same network as SCL:
   // ENO of a box is taken as its EN; it also drops when the box reports an error
   IF (#REQ_Open OR #REQ_Close) AND NOT #CMD.Sim AND "pulse_1s" THEN
       #OpTime_s := #OpTime_s + DINT#1;
       #OpTime_h := #OpTime_s / DINT#3600;
   END_IF;
END_REGION

REGION Network 34: Ограничение положения, мертвая зона
   RUNG wire#powerrail
      { S7_Templates := "SrcType := Real" } LT_Contact(in1 := #POSITION, in2 := #Pos_MIN)
      Move(in := #Pos_MIN, out1 => #POSITION)
   END_RUNG
   RUNG wire#powerrail
      { S7_Templates := "SrcType := Real" } GT_Contact(in1 := #POSITION, in2 := #Pos_MAX)
      Move(in := #Pos_MAX, out1 => #POSITION)
   END_RUNG
   RUNG wire#powerrail
      Add(in1 := #SP_M, in2 := #DB, out => #max)
      Sub(in1 := #SP_M, in2 := #DB, out => #min)
   END_RUNG
   // the same network as SCL:
   IF #POSITION < #Pos_MIN THEN #POSITION := #Pos_MIN; END_IF;
   IF #POSITION > #Pos_MAX THEN #POSITION := #Pos_MAX; END_IF;
   #max := #SP_M + #DB;
   #min := #SP_M - #DB;
END_REGION

REGION Network 35: Калибровка
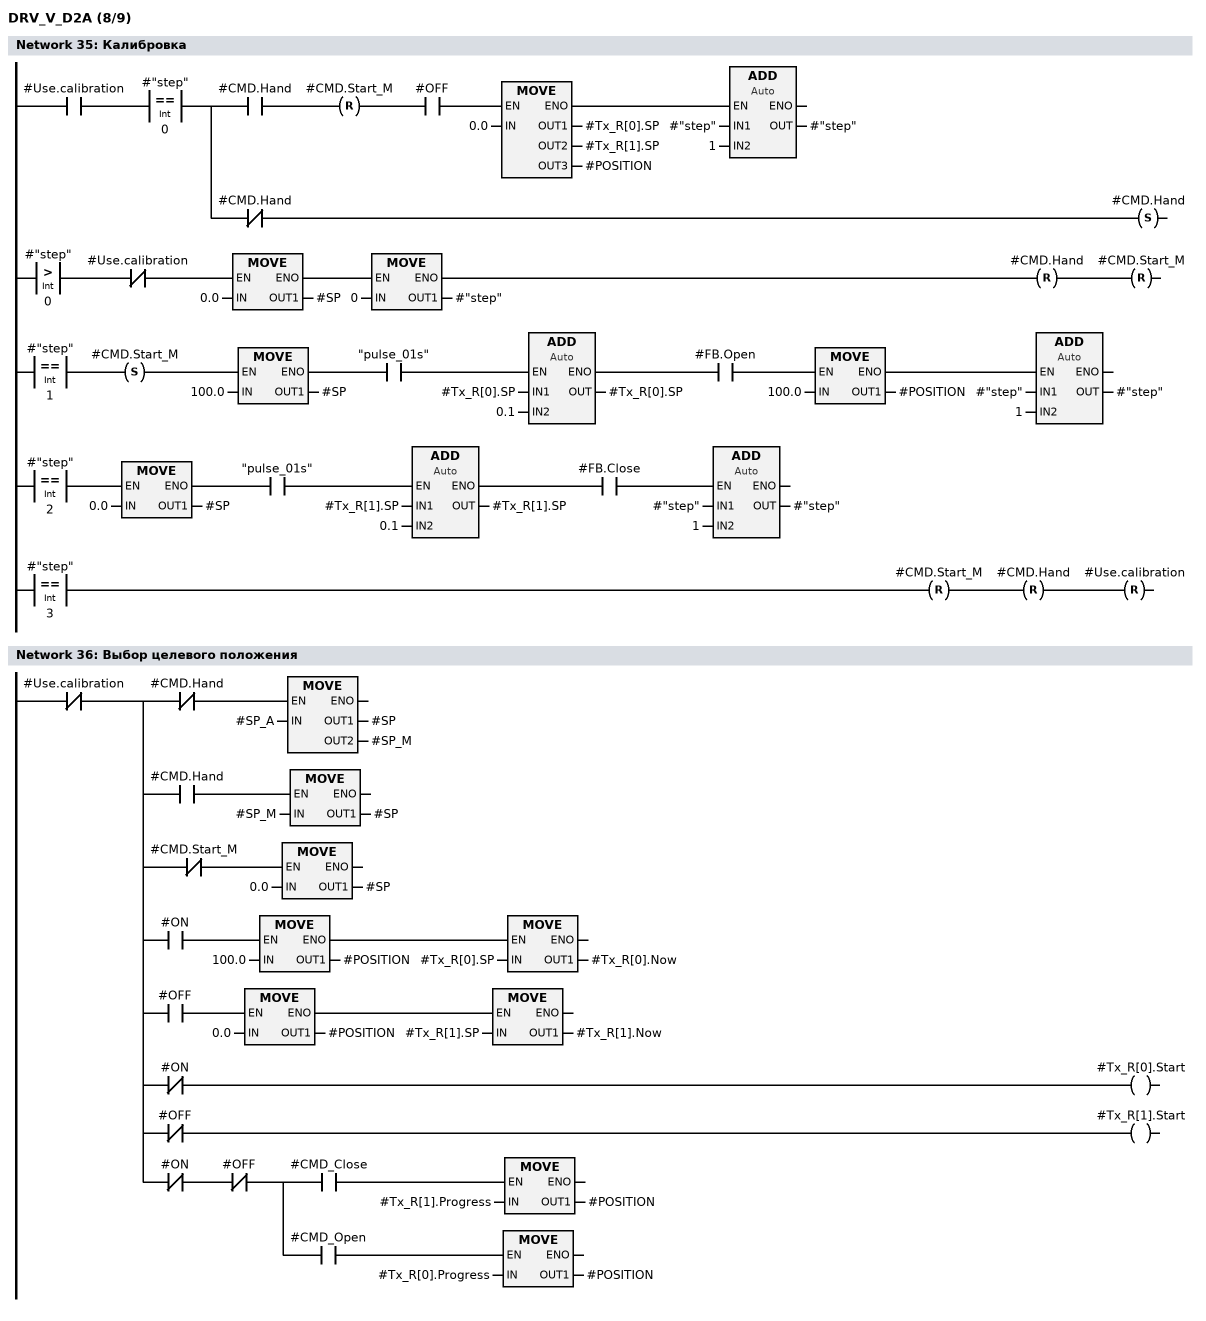
   RUNG wire#powerrail
      Contact( #Use.calibration )
      { S7_Templates := "SrcType := Int" } EQ_Contact(in1 := #"step", in2 := 0)
      wire#w1
      Contact( #CMD.Hand )
      R_Coil( #CMD.Start_M )
      Contact( #OFF )
      Move(in := 0.0, out1 => #Tx_R[0].SP, out2 => #Tx_R[1].SP, out3 => #POSITION)
      Add(in1 := #"step", in2 := 1, out => #"step")
   END_RUNG
   RUNG wire#w1
      I_Contact( #CMD.Hand )
      S_Coil( #CMD.Hand )
   END_RUNG
   RUNG wire#powerrail
      { S7_Templates := "SrcType := Int" } GT_Contact(in1 := #"step", in2 := 0)
      I_Contact( #Use.calibration )
      Move(in := 0.0, out1 => #SP)
      Move(in := 0, out1 => #"step")
      R_Coil( #CMD.Hand )
      R_Coil( #CMD.Start_M )
   END_RUNG
   RUNG wire#powerrail
      { S7_Templates := "SrcType := Int" } EQ_Contact(in1 := #"step", in2 := 1)
      S_Coil( #CMD.Start_M )
      Move(in := 100.0, out1 => #SP)
      Contact( "pulse_01s" )
      Add(in1 := #Tx_R[0].SP, in2 := 0.1, out => #Tx_R[0].SP)
      Contact( #FB.Open )
      Move(in := 100.0, out1 => #POSITION)
      Add(in1 := #"step", in2 := 1, out => #"step")
   END_RUNG
   RUNG wire#powerrail
      { S7_Templates := "SrcType := Int" } EQ_Contact(in1 := #"step", in2 := 2)
      Move(in := 0.0, out1 => #SP)
      Contact( "pulse_01s" )
      Add(in1 := #Tx_R[1].SP, in2 := 0.1, out => #Tx_R[1].SP)
      Contact( #FB.Close )
      Add(in1 := #"step", in2 := 1, out => #"step")
   END_RUNG
   RUNG wire#powerrail
      { S7_Templates := "SrcType := Int" } EQ_Contact(in1 := #"step", in2 := 3)
      R_Coil( #CMD.Start_M )
      R_Coil( #CMD.Hand )
      R_Coil( #Use.calibration )
   END_RUNG
   // the same network as SCL:
   #_w1 := #Use.calibration AND (#"step" = 0);
   #_w2 := #_w1 AND #CMD.Hand;
   IF #_w2 THEN #CMD.Start_M := FALSE; END_IF;
   IF #_w2 AND #OFF THEN
       #Tx_R[0].SP := 0.0;
       #Tx_R[1].SP := 0.0;
       #POSITION := 0.0;
       #"step" := #"step" + 1;
   END_IF;
   IF #_w1 AND NOT #CMD.Hand THEN #CMD.Hand := TRUE; END_IF;
   IF (#"step" > 0) AND NOT #Use.calibration THEN #SP := 0.0; END_IF;
   #_w3 := (#"step" > 0) AND NOT #Use.calibration;
   IF #_w3 THEN
       #"step" := 0;
       #CMD.Hand := FALSE;
       #CMD.Start_M := FALSE;
   END_IF;
   #_w4 := #"step" = 1;
   IF #_w4 THEN
       #CMD.Start_M := TRUE;
       #SP := 100.0;
   END_IF;
   #_w5 := #_w4 AND "pulse_01s";
   IF #_w5 THEN #Tx_R[0].SP := #Tx_R[0].SP + 0.1; END_IF;
   IF #_w5 AND #FB.Open THEN
       #POSITION := 100.0;
       #"step" := #"step" + 1;
   END_IF;
   #_w6 := #"step" = 2;
   IF #_w6 THEN #SP := 0.0; END_IF;
   #_w7 := #_w6 AND "pulse_01s";
   IF #_w7 THEN #Tx_R[1].SP := #Tx_R[1].SP + 0.1; END_IF;
   IF #_w7 AND #FB.Close THEN #"step" := #"step" + 1; END_IF;
   IF #"step" = 3 THEN
       #CMD.Start_M := FALSE;
       #CMD.Hand := FALSE;
       #Use.calibration := FALSE;
   END_IF;
END_REGION

REGION Network 36: Выбор целевого положения
   RUNG wire#powerrail
      I_Contact( #Use.calibration )
      wire#w1
      I_Contact( #CMD.Hand )
      Move(in := #SP_A, out1 => #SP, out2 => #SP_M)
   END_RUNG
   RUNG wire#w1
      Contact( #CMD.Hand )
      Move(in := #SP_M, out1 => #SP)
   END_RUNG
   RUNG wire#w1
      I_Contact( #CMD.Start_M )
      Move(in := 0.0, out1 => #SP)
   END_RUNG
   RUNG wire#w1
      Contact( #ON )
      Move(in := 100.0, out1 => #POSITION)
      Move(in := #Tx_R[0].SP, out1 => #Tx_R[0].Now)
   END_RUNG
   RUNG wire#w1
      Contact( #OFF )
      Move(in := 0.0, out1 => #POSITION)
      Move(in := #Tx_R[1].SP, out1 => #Tx_R[1].Now)
   END_RUNG
   RUNG wire#w1
      I_Contact( #ON )
      Coil( #Tx_R[0].Start )
   END_RUNG
   RUNG wire#w1
      I_Contact( #OFF )
      Coil( #Tx_R[1].Start )
   END_RUNG
   RUNG wire#w1
      I_Contact( #ON )
      I_Contact( #OFF )
      wire#w2
      Contact( #CMD_Close )
      Move(in := #Tx_R[1].Progress, out1 => #POSITION)
   END_RUNG
   RUNG wire#w2
      Contact( #CMD_Open )
      Move(in := #Tx_R[0].Progress, out1 => #POSITION)
   END_RUNG
   // the same network as SCL:
   IF NOT #Use.calibration AND NOT #CMD.Hand THEN
       #SP := #SP_A;
       #SP_M := #SP_A;
   END_IF;
   IF NOT #Use.calibration AND #CMD.Hand THEN #SP := #SP_M; END_IF;
   IF NOT #Use.calibration AND NOT #CMD.Start_M THEN #SP := 0.0; END_IF;
   IF NOT #Use.calibration AND #ON THEN
       #POSITION := 100.0;
       #Tx_R[0].Now := #Tx_R[0].SP;
   END_IF;
   IF NOT #Use.calibration AND #OFF THEN
       #POSITION := 0.0;
       #Tx_R[1].Now := #Tx_R[1].SP;
   END_IF;
   #Tx_R[0].Start := NOT #Use.calibration AND NOT #ON;
   #Tx_R[1].Start := NOT #Use.calibration AND NOT #OFF;
   #_w1 := NOT #Use.calibration AND NOT #ON AND NOT #OFF;
   IF #_w1 AND #CMD_Close THEN #POSITION := #Tx_R[1].Progress; END_IF;
   IF #_w1 AND #CMD_Open THEN #POSITION := #Tx_R[0].Progress; END_IF;
END_REGION

REGION Network 37: Определение текущего положения и команды
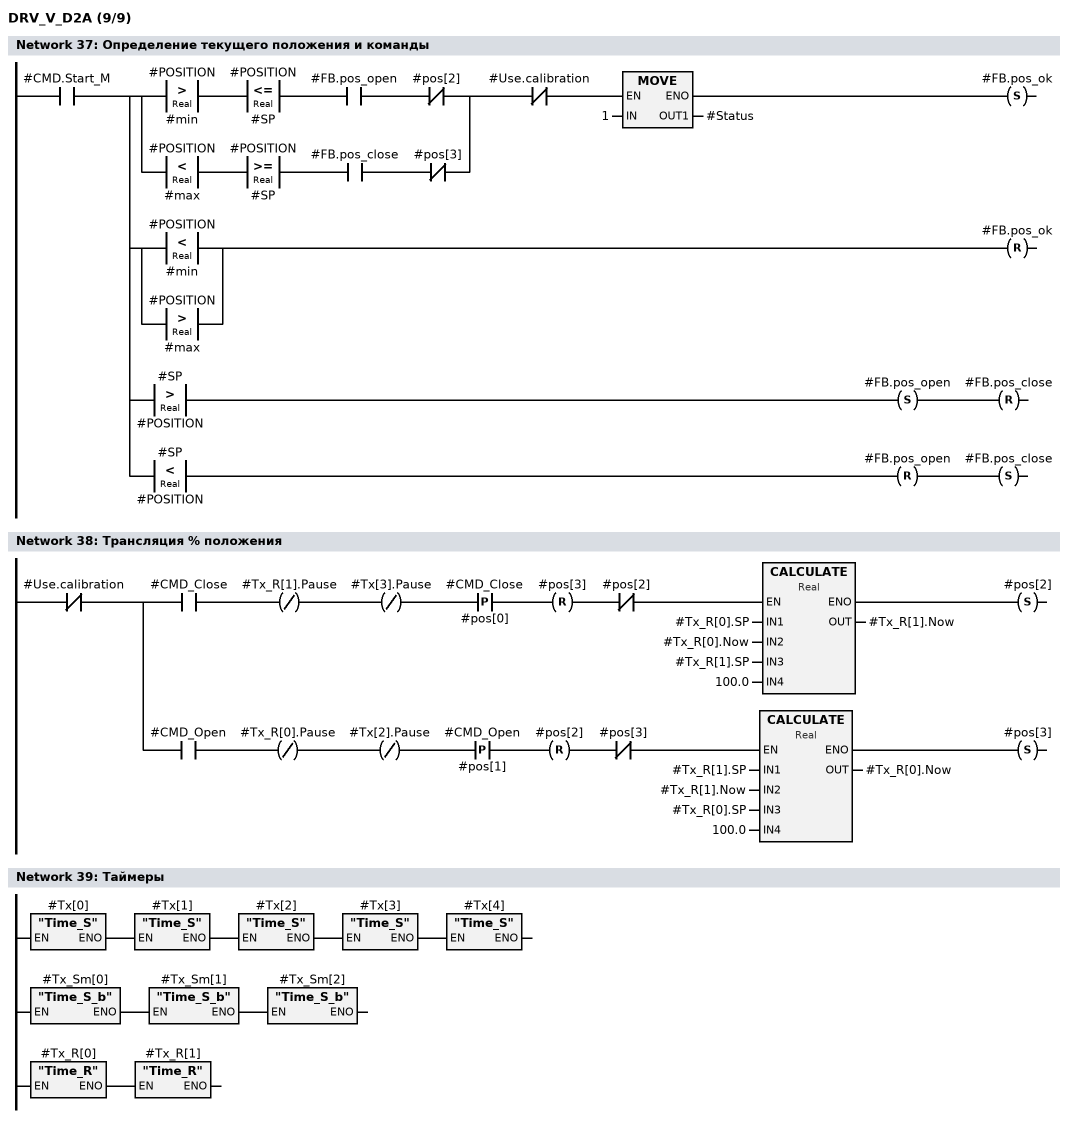
   RUNG wire#powerrail
      Contact( #CMD.Start_M )
      wire#w1
      { S7_Templates := "SrcType := Real" } GT_Contact(in1 := #POSITION, in2 := #min)
      { S7_Templates := "SrcType := Real" } LE_Contact(in1 := #POSITION, in2 := #SP)
      Contact( #FB.pos_open )
      I_Contact( #pos[2] )
      wire#w2
      I_Contact( #Use.calibration )
      Move(in := 1, out1 => #Status)
      S_Coil( #FB.pos_ok )
   END_RUNG
   RUNG wire#w1
      { S7_Templates := "SrcType := Real" } LT_Contact(in1 := #POSITION, in2 := #max)
      { S7_Templates := "SrcType := Real" } GE_Contact(in1 := #POSITION, in2 := #SP)
      Contact( #FB.pos_close )
      I_Contact( #pos[3] )
   END_RUNG wire#w2
   RUNG wire#w1
      { S7_Templates := "SrcType := Real" } LT_Contact(in1 := #POSITION, in2 := #min)
      wire#w3
      R_Coil( #FB.pos_ok )
   END_RUNG
   RUNG wire#w1
      { S7_Templates := "SrcType := Real" } GT_Contact(in1 := #POSITION, in2 := #max)
   END_RUNG wire#w3
   RUNG wire#w1
      { S7_Templates := "SrcType := Real" } GT_Contact(in1 := #SP, in2 := #POSITION)
      S_Coil( #FB.pos_open )
      R_Coil( #FB.pos_close )
   END_RUNG
   RUNG wire#w1
      { S7_Templates := "SrcType := Real" } LT_Contact(in1 := #SP, in2 := #POSITION)
      R_Coil( #FB.pos_open )
      S_Coil( #FB.pos_close )
   END_RUNG
   // the same network as SCL:
   IF #CMD.Start_M AND (((#POSITION > #min) AND (#POSITION <= #SP) AND #FB.pos_open AND NOT #pos[2]) OR ((#POSITION < #max) AND (#POSITION >= #SP) AND #FB.pos_close AND NOT #pos[3])) AND NOT #Use.calibration THEN
       #Status := 1;
       #FB.pos_ok := TRUE;
   END_IF;
   IF #CMD.Start_M AND ((#POSITION < #min) OR (#POSITION > #max)) THEN #FB.pos_ok := FALSE; END_IF;
   IF #CMD.Start_M AND (#SP > #POSITION) THEN
       #FB.pos_open := TRUE;
       #FB.pos_close := FALSE;
   END_IF;
   IF #CMD.Start_M AND (#SP < #POSITION) THEN
       #FB.pos_open := FALSE;
       #FB.pos_close := TRUE;
   END_IF;
END_REGION

REGION Network 38: Трансляция % положения
   RUNG wire#powerrail
      I_Contact( #Use.calibration )
      wire#w1
      Contact( #CMD_Close )
      I_Coil( #Tx_R[1].Pause )
      I_Coil( #Tx[3].Pause )
      P_Contact(operand := #CMD_Close, bit := #pos[0])
      R_Coil( #pos[3] )
      I_Contact( #pos[2] )
      { S7_Templates := "SrcType := Real"; S7_Expression := "(IN2/(IN1/IN4))*(IN3/IN4)" } Calculate(in1 := #Tx_R[0].SP, in2 := #Tx_R[0].Now, in3 := #Tx_R[1].SP, in4 := 100.0, out => #Tx_R[1].Now)
      S_Coil( #pos[2] )
   END_RUNG
   RUNG wire#w1
      Contact( #CMD_Open )
      I_Coil( #Tx_R[0].Pause )
      I_Coil( #Tx[2].Pause )
      P_Contact(operand := #CMD_Open, bit := #pos[1])
      R_Coil( #pos[2] )
      I_Contact( #pos[3] )
      { S7_Templates := "SrcType := Real"; S7_Expression := "(IN2/(IN1/IN4))*(IN3/IN4)" } Calculate(in1 := #Tx_R[1].SP, in2 := #Tx_R[1].Now, in3 := #Tx_R[0].SP, in4 := 100.0, out => #Tx_R[0].Now)
      S_Coil( #pos[3] )
   END_RUNG
   // the same network as SCL:
   #_w1 := NOT #Use.calibration AND #CMD_Close;
   #Tx_R[1].Pause := NOT #_w1;
   #Tx[3].Pause := NOT #_w1;
   #_w2 := #_w1 AND #CMD_Close AND NOT #pos[0];   // rising edge of #CMD_Close
   #pos[0] := #CMD_Close;
   IF #_w2 THEN #pos[3] := FALSE; END_IF;
   IF #_w2 AND NOT #pos[2] THEN
       #Tx_R[1].Now := (#Tx_R[0].Now/(#Tx_R[0].SP/100.0))*(#Tx_R[1].SP/100.0);
       #pos[2] := TRUE;
   END_IF;
   #_w3 := NOT #Use.calibration AND #CMD_Open;
   #Tx_R[0].Pause := NOT #_w3;
   #Tx[2].Pause := NOT #_w3;
   #_w4 := #_w3 AND #CMD_Open AND NOT #pos[1];   // rising edge of #CMD_Open
   #pos[1] := #CMD_Open;
   IF #_w4 THEN #pos[2] := FALSE; END_IF;
   IF #_w4 AND NOT #pos[3] THEN
       #Tx_R[0].Now := (#Tx_R[1].Now/(#Tx_R[1].SP/100.0))*(#Tx_R[0].SP/100.0);
       #pos[3] := TRUE;
   END_IF;
END_REGION

REGION Network 39: Таймеры
   RUNG wire#powerrail
      #Tx[0]()
      #Tx[1]()
      #Tx[2]()
      #Tx[3]()
      #Tx[4]()
   END_RUNG
   RUNG wire#powerrail
      #Tx_Sm[0]()
      #Tx_Sm[1]()
      #Tx_Sm[2]()
   END_RUNG
   RUNG wire#powerrail
      #Tx_R[0]()
      #Tx_R[1]()
   END_RUNG
   // the same network as SCL:
   #Tx[0](ENO => #_w1);   // "Time_S"
   #Tx[1](EN := #_w1, ENO => #_w2);   // "Time_S"
   #Tx[2](EN := #_w2, ENO => #_w3);   // "Time_S"
   #Tx[3](EN := #_w3, ENO => #_w4);   // "Time_S"
   IF #_w4 THEN
       #Tx[4]();   // "Time_S"
   END_IF;
   #Tx_Sm[0](ENO => #_w5);   // "Time_S_b"
   #Tx_Sm[1](EN := #_w5, ENO => #_w6);   // "Time_S_b"
   IF #_w6 THEN
       #Tx_Sm[2]();   // "Time_S_b"
   END_IF;
   #Tx_R[0](ENO => #_w7);   // "Time_R"
   IF #_w7 THEN
       #Tx_R[1]();   // "Time_R"
   END_IF;
END_REGION
END_FUNCTION_BLOCK
